// SIMATIC S7-200 project (STEP 7-Micro/WIN), CPU 224XP REL 02.01

ORGANIZATION_BLOCK PRINCIPAL:OB1
TITLE=COMENTARIOS DEL PROGRAMA
BEGIN
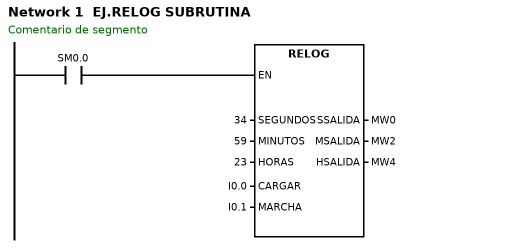
Network 1 // EJ.RELOG SUBRUTINA
// Comentario de segmento
LD     SM0.0
CALL   RELOG:SBR0, 34, 59, 23, I0.0, I0.1, MW0, MW2, MW4
END_ORGANIZATION_BLOCK

SUBROUTINE_BLOCK RELOG:SBR0
TITLE=COMENTARIOS DE LA SUBRUTINA
VAR_INPUT
SEGUNDOS:INT;	// LW0 
MINUTOS:INT;	// LW2 
HORAS:INT;	// LW4 
CARGAR:BOOL;	// L6.0 
MARCHA:BOOL;	// L6.1 
END_VAR
VAR_OUTPUT
SSALIDA:INT;	// LW7 
MSALIDA:INT;	// LW9 
HSALIDA:INT;	// LW11 
END_VAR
VAR
CSEGUNDO:INT;	// LW13 
CMINUTOS:INT;	// LW15 
CHORAS:INT;	// LW17 
END_VAR
BEGIN
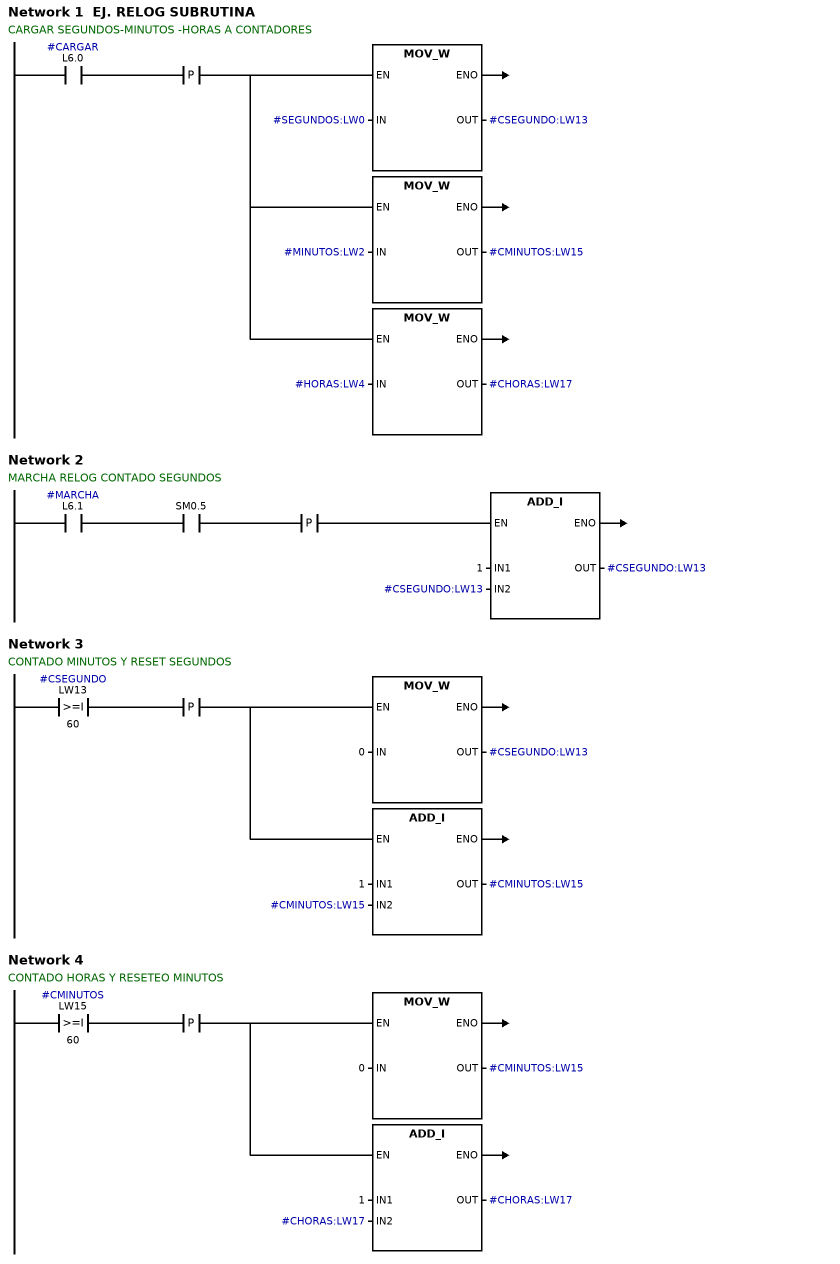
Network 1 // EJ. RELOG SUBRUTINA
// CARGAR SEGUNDOS-MINUTOS -HORAS A CONTADORES
LD     #CARGAR:L6.0
EU
MOVW   #SEGUNDOS:LW0, #CSEGUNDO:LW13
MOVW   #MINUTOS:LW2, #CMINUTOS:LW15
MOVW   #HORAS:LW4, #CHORAS:LW17
Network 2
// MARCHA RELOG CONTADO SEGUNDOS
LD     #MARCHA:L6.1
A      SM0.5
EU
+I     1, #CSEGUNDO:LW13
Network 3
// CONTADO MINUTOS Y RESET SEGUNDOS
LDW>=  #CSEGUNDO:LW13, 60
EU
MOVW   0, #CSEGUNDO:LW13
+I     1, #CMINUTOS:LW15
Network 4
// CONTADO HORAS Y RESETEO MINUTOS
LDW>=  #CMINUTOS:LW15, 60
EU
MOVW   0, #CMINUTOS:LW15
+I     1, #CHORAS:LW17
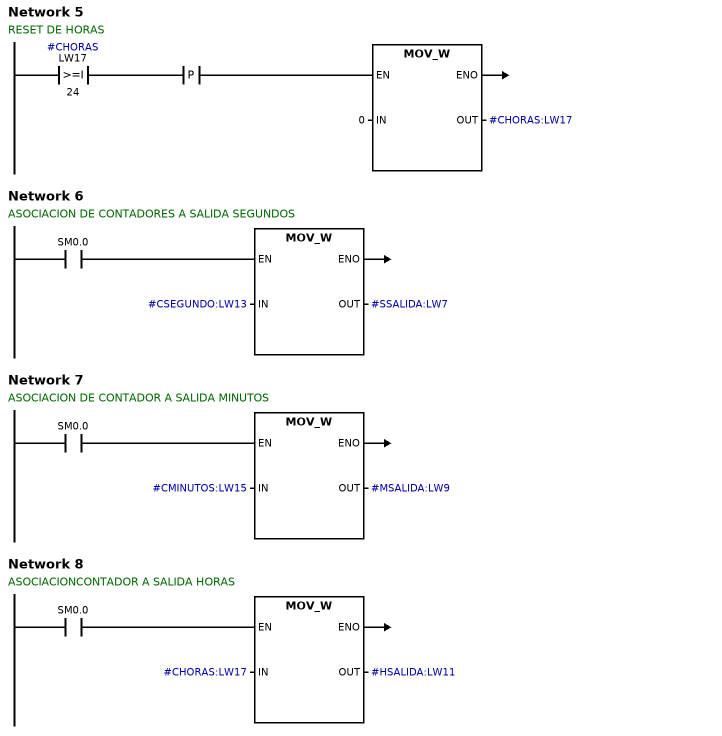
Network 5
// RESET DE HORAS 
LDW>=  #CHORAS:LW17, 24
EU
MOVW   0, #CHORAS:LW17
Network 6
// ASOCIACION DE CONTADORES A SALIDA SEGUNDOS
LD     SM0.0
MOVW   #CSEGUNDO:LW13, #SSALIDA:LW7
Network 7
// ASOCIACION DE CONTADOR A SALIDA MINUTOS
LD     SM0.0
MOVW   #CMINUTOS:LW15, #MSALIDA:LW9
Network 8
// ASOCIACIONCONTADOR A SALIDA HORAS
LD     SM0.0
MOVW   #CHORAS:LW17, #HSALIDA:LW11
END_SUBROUTINE_BLOCK
